// TIA Portal V20 export
TYPE "typeCmControlNodeInterlock"
// stored: Namespace Unit1.Em7
   STRUCT
      ngKicker { ExternalWritable := 'False'} : "LER_typeAxisInterlock";
      passKicker { ExternalWritable := 'False'} : "LER_typeAxisInterlock";
      cutConveyor { ExternalWritable := 'False'} : "LER_typeAxisInterlock";
      ngConveyor { ExternalWritable := 'False'} : "LER_typeAxisInterlock";
      stack1Conveyor { ExternalWritable := 'False'} : "LER_typeAxisInterlock";
      stack2Conveyor { ExternalWritable := 'False'} : "LER_typeAxisInterlock";
      conveyorVirtual { ExternalWritable := 'False'} : "LER_typeAxisInterlock";
      ngBoxLockCylinder { ExternalWritable := 'False'} : "LER_typeTwoWayActuatorInterlock";
   END_STRUCT;
END_TYPE
